PROGRAM PRG_BuyCoffee
VAR
END_VAR

END_PROGRAM

(* stored: Version 1.1.0.1, ProductVersion 3.1.4024.15
   POU PRG_BuyCoffee: Id {9a6699d9-b0d8-4795-a2c4-9a9be7bf6a9a}, SpecialFunc None *)
